PROGRAM MAIN
VAR
	output2 AT %Q* : BOOL;
END_VAR

END_PROGRAM

(* stored: Version 1.1.0.1, ProductVersion 3.1.4024.2
   POU MAIN: Id {faf86287-4e03-44c8-867a-c0b2a97e9a66}, SpecialFunc None *)
